// TIA Portal V17 export
// export: Created 2025-05-22T05:59:42.0139145Z, ExportSetting WithDefaults, DisplayName Totally Integrated Automation Portal, DisplayVersion V17 Update 8, DisplayName TIA Portal Openness, DisplayVersion V17 Update 8, DisplayName TIA Portal Version Control Interface, DisplayVersion V17, DisplayName SINAMICS Startdrive Advanced, DisplayVersion V17 SP2, DisplayName SINAMICS Startdrive G110M, G120, G120C, G120D, G120P, G115D, DisplayVersion V17 SP2, DisplayName SINAMICS Startdrive G130, G150, S120, S150, SINAMICS MV, S210, DisplayVersion V17 SP2, DisplayName STEP 7 Professional, DisplayVersion V17 Update 8, DisplayName SINUMERIK ONE STEP 7 Toolbox, DisplayVersion V17 Update 12, DisplayName SINUMERIK ONE PLC Basic Program Plus, DisplayVersion V17 Update 12, DisplayName SINUMERIK 840D sl STEP 7 Toolbox, DisplayVersion V17 Update 12, DisplayName STEP 7 Safety, DisplayVersion V17 Update 6, DisplayName WinCC Advanced, DisplayVersion V17 Update 8
FUNCTION "FC4001_JAW_CHUCK_CONTROL_U2_STA_1" : Void   // FC4001, LAD
{ S7_Optimized_Access := 'TRUE' }
VERSION : 0.1
// stored: AutoNumber false, IsIECCheckEnabled false, SetENOAutomatically false, UDAEnableTagReadback false
   VAR_TEMP
      TEMP_SENSOR_VALUE_1 : UInt;
      TEMP_SENSOR_VALUE : UInt;
   END_VAR
BEGIN

REGION Network 1
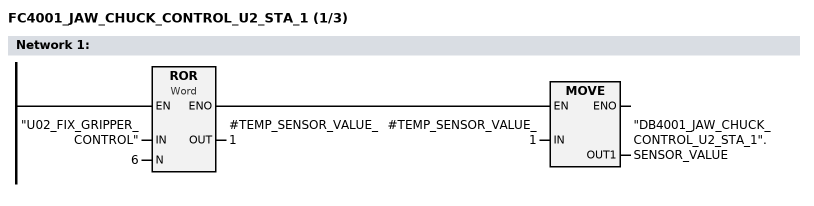
   #TEMP_SENSOR_VALUE_1 := ROR(IN := "U02_FIX_GRIPPER_CONTROL", N := 6);
   "DB4001_JAW_CHUCK_CONTROL_U2_STA_1".SENSOR_VALUE := #TEMP_SENSOR_VALUE_1;
END_REGION

REGION Network 2: UNIT 01 STATION 1 FIXTURE CLAMPED
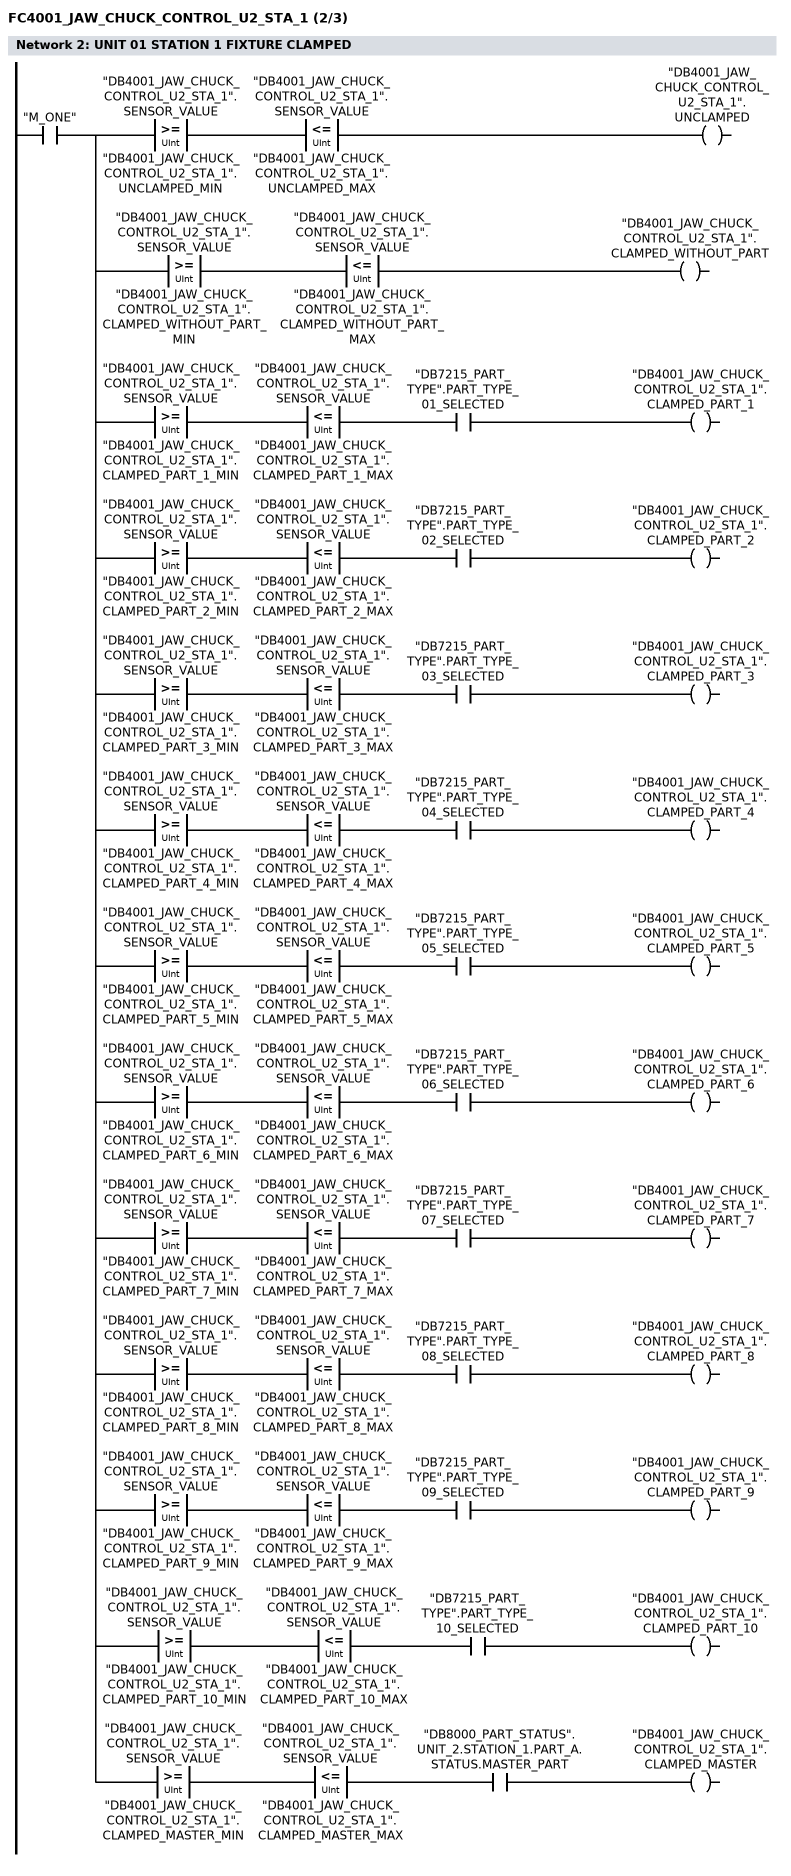
   RUNG wire#powerrail
      Contact( "M_ONE" )
      wire#w1
      { S7_Templates := "SrcType := UInt" } GE_Contact(in1 := "DB4001_JAW_CHUCK_CONTROL_U2_STA_1".SENSOR_VALUE, in2 := "DB4001_JAW_CHUCK_CONTROL_U2_STA_1".UNCLAMPED_MIN)
      { S7_Templates := "SrcType := UInt" } LE_Contact(in1 := "DB4001_JAW_CHUCK_CONTROL_U2_STA_1".SENSOR_VALUE, in2 := "DB4001_JAW_CHUCK_CONTROL_U2_STA_1".UNCLAMPED_MAX)
      Coil( "DB4001_JAW_CHUCK_CONTROL_U2_STA_1".UNCLAMPED )
   END_RUNG
   RUNG wire#w1
      { S7_Templates := "SrcType := UInt" } GE_Contact(in1 := "DB4001_JAW_CHUCK_CONTROL_U2_STA_1".SENSOR_VALUE, in2 := "DB4001_JAW_CHUCK_CONTROL_U2_STA_1".CLAMPED_WITHOUT_PART_MIN)
      { S7_Templates := "SrcType := UInt" } LE_Contact(in1 := "DB4001_JAW_CHUCK_CONTROL_U2_STA_1".SENSOR_VALUE, in2 := "DB4001_JAW_CHUCK_CONTROL_U2_STA_1".CLAMPED_WITHOUT_PART_MAX)
      Coil( "DB4001_JAW_CHUCK_CONTROL_U2_STA_1".CLAMPED_WITHOUT_PART )
   END_RUNG
   RUNG wire#w1
      { S7_Templates := "SrcType := UInt" } GE_Contact(in1 := "DB4001_JAW_CHUCK_CONTROL_U2_STA_1".SENSOR_VALUE, in2 := "DB4001_JAW_CHUCK_CONTROL_U2_STA_1".CLAMPED_PART_1_MIN)
      { S7_Templates := "SrcType := UInt" } LE_Contact(in1 := "DB4001_JAW_CHUCK_CONTROL_U2_STA_1".SENSOR_VALUE, in2 := "DB4001_JAW_CHUCK_CONTROL_U2_STA_1".CLAMPED_PART_1_MAX)
      Contact( "DB7215_PART_TYPE".PART_TYPE_01_SELECTED )
      Coil( "DB4001_JAW_CHUCK_CONTROL_U2_STA_1".CLAMPED_PART_1 )
   END_RUNG
   RUNG wire#w1
      { S7_Templates := "SrcType := UInt" } GE_Contact(in1 := "DB4001_JAW_CHUCK_CONTROL_U2_STA_1".SENSOR_VALUE, in2 := "DB4001_JAW_CHUCK_CONTROL_U2_STA_1".CLAMPED_PART_2_MIN)
      { S7_Templates := "SrcType := UInt" } LE_Contact(in1 := "DB4001_JAW_CHUCK_CONTROL_U2_STA_1".SENSOR_VALUE, in2 := "DB4001_JAW_CHUCK_CONTROL_U2_STA_1".CLAMPED_PART_2_MAX)
      Contact( "DB7215_PART_TYPE".PART_TYPE_02_SELECTED )
      Coil( "DB4001_JAW_CHUCK_CONTROL_U2_STA_1".CLAMPED_PART_2 )
   END_RUNG
   RUNG wire#w1
      { S7_Templates := "SrcType := UInt" } GE_Contact(in1 := "DB4001_JAW_CHUCK_CONTROL_U2_STA_1".SENSOR_VALUE, in2 := "DB4001_JAW_CHUCK_CONTROL_U2_STA_1".CLAMPED_PART_3_MIN)
      { S7_Templates := "SrcType := UInt" } LE_Contact(in1 := "DB4001_JAW_CHUCK_CONTROL_U2_STA_1".SENSOR_VALUE, in2 := "DB4001_JAW_CHUCK_CONTROL_U2_STA_1".CLAMPED_PART_3_MAX)
      Contact( "DB7215_PART_TYPE".PART_TYPE_03_SELECTED )
      Coil( "DB4001_JAW_CHUCK_CONTROL_U2_STA_1".CLAMPED_PART_3 )
   END_RUNG
   RUNG wire#w1
      { S7_Templates := "SrcType := UInt" } GE_Contact(in1 := "DB4001_JAW_CHUCK_CONTROL_U2_STA_1".SENSOR_VALUE, in2 := "DB4001_JAW_CHUCK_CONTROL_U2_STA_1".CLAMPED_PART_4_MIN)
      { S7_Templates := "SrcType := UInt" } LE_Contact(in1 := "DB4001_JAW_CHUCK_CONTROL_U2_STA_1".SENSOR_VALUE, in2 := "DB4001_JAW_CHUCK_CONTROL_U2_STA_1".CLAMPED_PART_4_MAX)
      Contact( "DB7215_PART_TYPE".PART_TYPE_04_SELECTED )
      Coil( "DB4001_JAW_CHUCK_CONTROL_U2_STA_1".CLAMPED_PART_4 )
   END_RUNG
   RUNG wire#w1
      { S7_Templates := "SrcType := UInt" } GE_Contact(in1 := "DB4001_JAW_CHUCK_CONTROL_U2_STA_1".SENSOR_VALUE, in2 := "DB4001_JAW_CHUCK_CONTROL_U2_STA_1".CLAMPED_PART_5_MIN)
      { S7_Templates := "SrcType := UInt" } LE_Contact(in1 := "DB4001_JAW_CHUCK_CONTROL_U2_STA_1".SENSOR_VALUE, in2 := "DB4001_JAW_CHUCK_CONTROL_U2_STA_1".CLAMPED_PART_5_MAX)
      Contact( "DB7215_PART_TYPE".PART_TYPE_05_SELECTED )
      Coil( "DB4001_JAW_CHUCK_CONTROL_U2_STA_1".CLAMPED_PART_5 )
   END_RUNG
   RUNG wire#w1
      { S7_Templates := "SrcType := UInt" } GE_Contact(in1 := "DB4001_JAW_CHUCK_CONTROL_U2_STA_1".SENSOR_VALUE, in2 := "DB4001_JAW_CHUCK_CONTROL_U2_STA_1".CLAMPED_PART_6_MIN)
      { S7_Templates := "SrcType := UInt" } LE_Contact(in1 := "DB4001_JAW_CHUCK_CONTROL_U2_STA_1".SENSOR_VALUE, in2 := "DB4001_JAW_CHUCK_CONTROL_U2_STA_1".CLAMPED_PART_6_MAX)
      Contact( "DB7215_PART_TYPE".PART_TYPE_06_SELECTED )
      Coil( "DB4001_JAW_CHUCK_CONTROL_U2_STA_1".CLAMPED_PART_6 )
   END_RUNG
   RUNG wire#w1
      { S7_Templates := "SrcType := UInt" } GE_Contact(in1 := "DB4001_JAW_CHUCK_CONTROL_U2_STA_1".SENSOR_VALUE, in2 := "DB4001_JAW_CHUCK_CONTROL_U2_STA_1".CLAMPED_PART_7_MIN)
      { S7_Templates := "SrcType := UInt" } LE_Contact(in1 := "DB4001_JAW_CHUCK_CONTROL_U2_STA_1".SENSOR_VALUE, in2 := "DB4001_JAW_CHUCK_CONTROL_U2_STA_1".CLAMPED_PART_7_MAX)
      Contact( "DB7215_PART_TYPE".PART_TYPE_07_SELECTED )
      Coil( "DB4001_JAW_CHUCK_CONTROL_U2_STA_1".CLAMPED_PART_7 )
   END_RUNG
   RUNG wire#w1
      { S7_Templates := "SrcType := UInt" } GE_Contact(in1 := "DB4001_JAW_CHUCK_CONTROL_U2_STA_1".SENSOR_VALUE, in2 := "DB4001_JAW_CHUCK_CONTROL_U2_STA_1".CLAMPED_PART_8_MIN)
      { S7_Templates := "SrcType := UInt" } LE_Contact(in1 := "DB4001_JAW_CHUCK_CONTROL_U2_STA_1".SENSOR_VALUE, in2 := "DB4001_JAW_CHUCK_CONTROL_U2_STA_1".CLAMPED_PART_8_MAX)
      Contact( "DB7215_PART_TYPE".PART_TYPE_08_SELECTED )
      Coil( "DB4001_JAW_CHUCK_CONTROL_U2_STA_1".CLAMPED_PART_8 )
   END_RUNG
   RUNG wire#w1
      { S7_Templates := "SrcType := UInt" } GE_Contact(in1 := "DB4001_JAW_CHUCK_CONTROL_U2_STA_1".SENSOR_VALUE, in2 := "DB4001_JAW_CHUCK_CONTROL_U2_STA_1".CLAMPED_PART_9_MIN)
      { S7_Templates := "SrcType := UInt" } LE_Contact(in1 := "DB4001_JAW_CHUCK_CONTROL_U2_STA_1".SENSOR_VALUE, in2 := "DB4001_JAW_CHUCK_CONTROL_U2_STA_1".CLAMPED_PART_9_MAX)
      Contact( "DB7215_PART_TYPE".PART_TYPE_09_SELECTED )
      Coil( "DB4001_JAW_CHUCK_CONTROL_U2_STA_1".CLAMPED_PART_9 )
   END_RUNG
   RUNG wire#w1
      { S7_Templates := "SrcType := UInt" } GE_Contact(in1 := "DB4001_JAW_CHUCK_CONTROL_U2_STA_1".SENSOR_VALUE, in2 := "DB4001_JAW_CHUCK_CONTROL_U2_STA_1".CLAMPED_PART_10_MIN)
      { S7_Templates := "SrcType := UInt" } LE_Contact(in1 := "DB4001_JAW_CHUCK_CONTROL_U2_STA_1".SENSOR_VALUE, in2 := "DB4001_JAW_CHUCK_CONTROL_U2_STA_1".CLAMPED_PART_10_MAX)
      Contact( "DB7215_PART_TYPE".PART_TYPE_10_SELECTED )
      Coil( "DB4001_JAW_CHUCK_CONTROL_U2_STA_1".CLAMPED_PART_10 )
   END_RUNG
   RUNG wire#w1
      { S7_Templates := "SrcType := UInt" } GE_Contact(in1 := "DB4001_JAW_CHUCK_CONTROL_U2_STA_1".SENSOR_VALUE, in2 := "DB4001_JAW_CHUCK_CONTROL_U2_STA_1".CLAMPED_MASTER_MIN)
      { S7_Templates := "SrcType := UInt" } LE_Contact(in1 := "DB4001_JAW_CHUCK_CONTROL_U2_STA_1".SENSOR_VALUE, in2 := "DB4001_JAW_CHUCK_CONTROL_U2_STA_1".CLAMPED_MASTER_MAX)
      Contact( "DB8000_PART_STATUS".UNIT_2.STATION_1.PART_A.STATUS.MASTER_PART )
      Coil( "DB4001_JAW_CHUCK_CONTROL_U2_STA_1".CLAMPED_MASTER )
   END_RUNG
   // the same network as SCL:
   "DB4001_JAW_CHUCK_CONTROL_U2_STA_1".UNCLAMPED := "M_ONE" AND ("DB4001_JAW_CHUCK_CONTROL_U2_STA_1".SENSOR_VALUE >= "DB4001_JAW_CHUCK_CONTROL_U2_STA_1".UNCLAMPED_MIN) AND ("DB4001_JAW_CHUCK_CONTROL_U2_STA_1".SENSOR_VALUE <= "DB4001_JAW_CHUCK_CONTROL_U2_STA_1".UNCLAMPED_MAX);
   "DB4001_JAW_CHUCK_CONTROL_U2_STA_1".CLAMPED_WITHOUT_PART := "M_ONE" AND ("DB4001_JAW_CHUCK_CONTROL_U2_STA_1".SENSOR_VALUE >= "DB4001_JAW_CHUCK_CONTROL_U2_STA_1".CLAMPED_WITHOUT_PART_MIN) AND ("DB4001_JAW_CHUCK_CONTROL_U2_STA_1".SENSOR_VALUE <= "DB4001_JAW_CHUCK_CONTROL_U2_STA_1".CLAMPED_WITHOUT_PART_MAX);
   "DB4001_JAW_CHUCK_CONTROL_U2_STA_1".CLAMPED_PART_1 := "M_ONE" AND ("DB4001_JAW_CHUCK_CONTROL_U2_STA_1".SENSOR_VALUE >= "DB4001_JAW_CHUCK_CONTROL_U2_STA_1".CLAMPED_PART_1_MIN) AND ("DB4001_JAW_CHUCK_CONTROL_U2_STA_1".SENSOR_VALUE <= "DB4001_JAW_CHUCK_CONTROL_U2_STA_1".CLAMPED_PART_1_MAX) AND "DB7215_PART_TYPE".PART_TYPE_01_SELECTED;
   "DB4001_JAW_CHUCK_CONTROL_U2_STA_1".CLAMPED_PART_2 := "M_ONE" AND ("DB4001_JAW_CHUCK_CONTROL_U2_STA_1".SENSOR_VALUE >= "DB4001_JAW_CHUCK_CONTROL_U2_STA_1".CLAMPED_PART_2_MIN) AND ("DB4001_JAW_CHUCK_CONTROL_U2_STA_1".SENSOR_VALUE <= "DB4001_JAW_CHUCK_CONTROL_U2_STA_1".CLAMPED_PART_2_MAX) AND "DB7215_PART_TYPE".PART_TYPE_02_SELECTED;
   "DB4001_JAW_CHUCK_CONTROL_U2_STA_1".CLAMPED_PART_3 := "M_ONE" AND ("DB4001_JAW_CHUCK_CONTROL_U2_STA_1".SENSOR_VALUE >= "DB4001_JAW_CHUCK_CONTROL_U2_STA_1".CLAMPED_PART_3_MIN) AND ("DB4001_JAW_CHUCK_CONTROL_U2_STA_1".SENSOR_VALUE <= "DB4001_JAW_CHUCK_CONTROL_U2_STA_1".CLAMPED_PART_3_MAX) AND "DB7215_PART_TYPE".PART_TYPE_03_SELECTED;
   "DB4001_JAW_CHUCK_CONTROL_U2_STA_1".CLAMPED_PART_4 := "M_ONE" AND ("DB4001_JAW_CHUCK_CONTROL_U2_STA_1".SENSOR_VALUE >= "DB4001_JAW_CHUCK_CONTROL_U2_STA_1".CLAMPED_PART_4_MIN) AND ("DB4001_JAW_CHUCK_CONTROL_U2_STA_1".SENSOR_VALUE <= "DB4001_JAW_CHUCK_CONTROL_U2_STA_1".CLAMPED_PART_4_MAX) AND "DB7215_PART_TYPE".PART_TYPE_04_SELECTED;
   "DB4001_JAW_CHUCK_CONTROL_U2_STA_1".CLAMPED_PART_5 := "M_ONE" AND ("DB4001_JAW_CHUCK_CONTROL_U2_STA_1".SENSOR_VALUE >= "DB4001_JAW_CHUCK_CONTROL_U2_STA_1".CLAMPED_PART_5_MIN) AND ("DB4001_JAW_CHUCK_CONTROL_U2_STA_1".SENSOR_VALUE <= "DB4001_JAW_CHUCK_CONTROL_U2_STA_1".CLAMPED_PART_5_MAX) AND "DB7215_PART_TYPE".PART_TYPE_05_SELECTED;
   "DB4001_JAW_CHUCK_CONTROL_U2_STA_1".CLAMPED_PART_6 := "M_ONE" AND ("DB4001_JAW_CHUCK_CONTROL_U2_STA_1".SENSOR_VALUE >= "DB4001_JAW_CHUCK_CONTROL_U2_STA_1".CLAMPED_PART_6_MIN) AND ("DB4001_JAW_CHUCK_CONTROL_U2_STA_1".SENSOR_VALUE <= "DB4001_JAW_CHUCK_CONTROL_U2_STA_1".CLAMPED_PART_6_MAX) AND "DB7215_PART_TYPE".PART_TYPE_06_SELECTED;
   "DB4001_JAW_CHUCK_CONTROL_U2_STA_1".CLAMPED_PART_7 := "M_ONE" AND ("DB4001_JAW_CHUCK_CONTROL_U2_STA_1".SENSOR_VALUE >= "DB4001_JAW_CHUCK_CONTROL_U2_STA_1".CLAMPED_PART_7_MIN) AND ("DB4001_JAW_CHUCK_CONTROL_U2_STA_1".SENSOR_VALUE <= "DB4001_JAW_CHUCK_CONTROL_U2_STA_1".CLAMPED_PART_7_MAX) AND "DB7215_PART_TYPE".PART_TYPE_07_SELECTED;
   "DB4001_JAW_CHUCK_CONTROL_U2_STA_1".CLAMPED_PART_8 := "M_ONE" AND ("DB4001_JAW_CHUCK_CONTROL_U2_STA_1".SENSOR_VALUE >= "DB4001_JAW_CHUCK_CONTROL_U2_STA_1".CLAMPED_PART_8_MIN) AND ("DB4001_JAW_CHUCK_CONTROL_U2_STA_1".SENSOR_VALUE <= "DB4001_JAW_CHUCK_CONTROL_U2_STA_1".CLAMPED_PART_8_MAX) AND "DB7215_PART_TYPE".PART_TYPE_08_SELECTED;
   "DB4001_JAW_CHUCK_CONTROL_U2_STA_1".CLAMPED_PART_9 := "M_ONE" AND ("DB4001_JAW_CHUCK_CONTROL_U2_STA_1".SENSOR_VALUE >= "DB4001_JAW_CHUCK_CONTROL_U2_STA_1".CLAMPED_PART_9_MIN) AND ("DB4001_JAW_CHUCK_CONTROL_U2_STA_1".SENSOR_VALUE <= "DB4001_JAW_CHUCK_CONTROL_U2_STA_1".CLAMPED_PART_9_MAX) AND "DB7215_PART_TYPE".PART_TYPE_09_SELECTED;
   "DB4001_JAW_CHUCK_CONTROL_U2_STA_1".CLAMPED_PART_10 := "M_ONE" AND ("DB4001_JAW_CHUCK_CONTROL_U2_STA_1".SENSOR_VALUE >= "DB4001_JAW_CHUCK_CONTROL_U2_STA_1".CLAMPED_PART_10_MIN) AND ("DB4001_JAW_CHUCK_CONTROL_U2_STA_1".SENSOR_VALUE <= "DB4001_JAW_CHUCK_CONTROL_U2_STA_1".CLAMPED_PART_10_MAX) AND "DB7215_PART_TYPE".PART_TYPE_10_SELECTED;
   "DB4001_JAW_CHUCK_CONTROL_U2_STA_1".CLAMPED_MASTER := "M_ONE" AND ("DB4001_JAW_CHUCK_CONTROL_U2_STA_1".SENSOR_VALUE >= "DB4001_JAW_CHUCK_CONTROL_U2_STA_1".CLAMPED_MASTER_MIN) AND ("DB4001_JAW_CHUCK_CONTROL_U2_STA_1".SENSOR_VALUE <= "DB4001_JAW_CHUCK_CONTROL_U2_STA_1".CLAMPED_MASTER_MAX) AND "DB8000_PART_STATUS".UNIT_2.STATION_1.PART_A.STATUS.MASTER_PART;
END_REGION

REGION Network 3: FIXTURE NOT CLAMPED TIME EXCEEDED ALARM
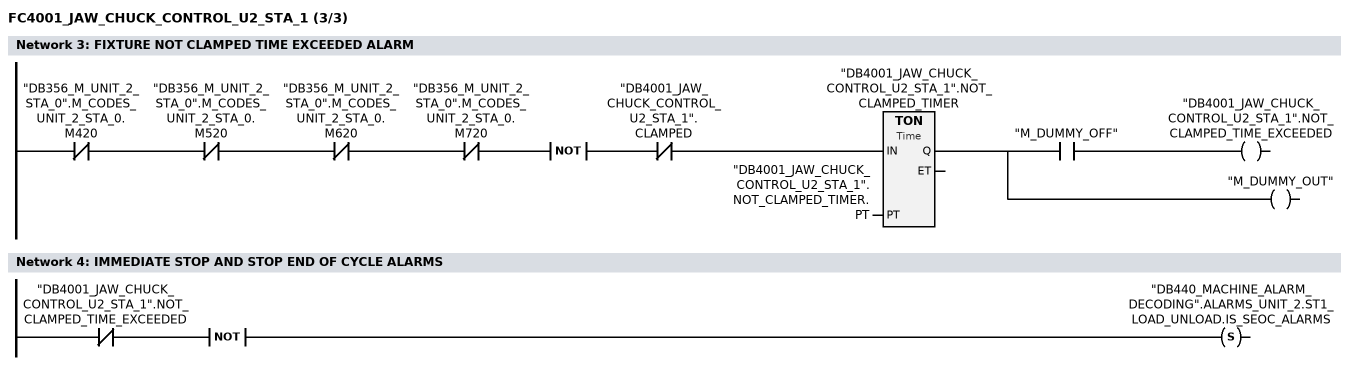
   RUNG wire#powerrail
      I_Contact( "DB356_M_UNIT_2_STA_0".M_CODES_UNIT_2_STA_0.M420 )
      I_Contact( "DB356_M_UNIT_2_STA_0".M_CODES_UNIT_2_STA_0.M520 )
      I_Contact( "DB356_M_UNIT_2_STA_0".M_CODES_UNIT_2_STA_0.M620 )
      I_Contact( "DB356_M_UNIT_2_STA_0".M_CODES_UNIT_2_STA_0.M720 )
      Not()
      I_Contact( "DB4001_JAW_CHUCK_CONTROL_U2_STA_1".CLAMPED )
      { S7_Templates := "time_type := Time" } "DB4001_JAW_CHUCK_CONTROL_U2_STA_1".NOT_CLAMPED_TIMER.TON(pt := "DB4001_JAW_CHUCK_CONTROL_U2_STA_1".NOT_CLAMPED_TIMER.PT, et =>)
      wire#w1
      Contact( "M_DUMMY_OFF" )
      Coil( "DB4001_JAW_CHUCK_CONTROL_U2_STA_1".NOT_CLAMPED_TIME_EXCEEDED )
   END_RUNG
   RUNG wire#w1
      Coil( "M_DUMMY_OUT" )
   END_RUNG
   // the same network as SCL:
   "DB4001_JAW_CHUCK_CONTROL_U2_STA_1".NOT_CLAMPED_TIMER.TON(IN := NOT (NOT "DB356_M_UNIT_2_STA_0".M_CODES_UNIT_2_STA_0.M420 AND NOT "DB356_M_UNIT_2_STA_0".M_CODES_UNIT_2_STA_0.M520 AND NOT "DB356_M_UNIT_2_STA_0".M_CODES_UNIT_2_STA_0.M620 AND NOT "DB356_M_UNIT_2_STA_0".M_CODES_UNIT_2_STA_0.M720) AND NOT "DB4001_JAW_CHUCK_CONTROL_U2_STA_1".CLAMPED,
                           PT := "DB4001_JAW_CHUCK_CONTROL_U2_STA_1".NOT_CLAMPED_TIMER.PT);
   "DB4001_JAW_CHUCK_CONTROL_U2_STA_1".NOT_CLAMPED_TIME_EXCEEDED := "DB4001_JAW_CHUCK_CONTROL_U2_STA_1".NOT_CLAMPED_TIMER.Q AND "M_DUMMY_OFF";
   "M_DUMMY_OUT" := "DB4001_JAW_CHUCK_CONTROL_U2_STA_1".NOT_CLAMPED_TIMER.Q;
END_REGION

REGION Network 4: IMMEDIATE STOP AND STOP END OF CYCLE ALARMS
   RUNG wire#powerrail
      I_Contact( "DB4001_JAW_CHUCK_CONTROL_U2_STA_1".NOT_CLAMPED_TIME_EXCEEDED )
      Not()
      S_Coil( "DB440_MACHINE_ALARM_DECODING".ALARMS_UNIT_2.ST1_LOAD_UNLOAD.IS_SEOC_ALARMS )
   END_RUNG
   // the same network as SCL:
   IF NOT (NOT "DB4001_JAW_CHUCK_CONTROL_U2_STA_1".NOT_CLAMPED_TIME_EXCEEDED) THEN
       "DB440_MACHINE_ALARM_DECODING".ALARMS_UNIT_2.ST1_LOAD_UNLOAD.IS_SEOC_ALARMS := TRUE;
   END_IF;
END_REGION
END_FUNCTION
